FUNCTION_BLOCK TransferUnit (* Composite Function Block Type *)
  (* Standard: 61499-2 *)
  (* Version 0.0, 7/14/2016, Andrei, nxtControl GmbH, template *)
  PACKAGE Main;
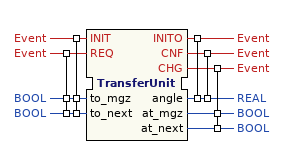
  EVENT_INPUT
    INIT WITH to_mgz, to_next; (* Initialization Request *)
    REQ WITH to_mgz, to_next; (* Normal Execution Request *)
  END_EVENT
  EVENT_OUTPUT
    INITO WITH angle; (* Initialization Confirm *)
    CNF WITH angle; (* Execution Confirmation *)
    CHG WITH at_mgz, at_next;
  END_EVENT
  VAR_INPUT
    to_mgz : BOOL; (* Input event qualifier *)
    to_next : BOOL;
  END_VAR
  VAR_OUTPUT
    angle : REAL; (* Output event qualifier *)
    at_mgz : BOOL;
    at_next : BOOL;
  END_VAR
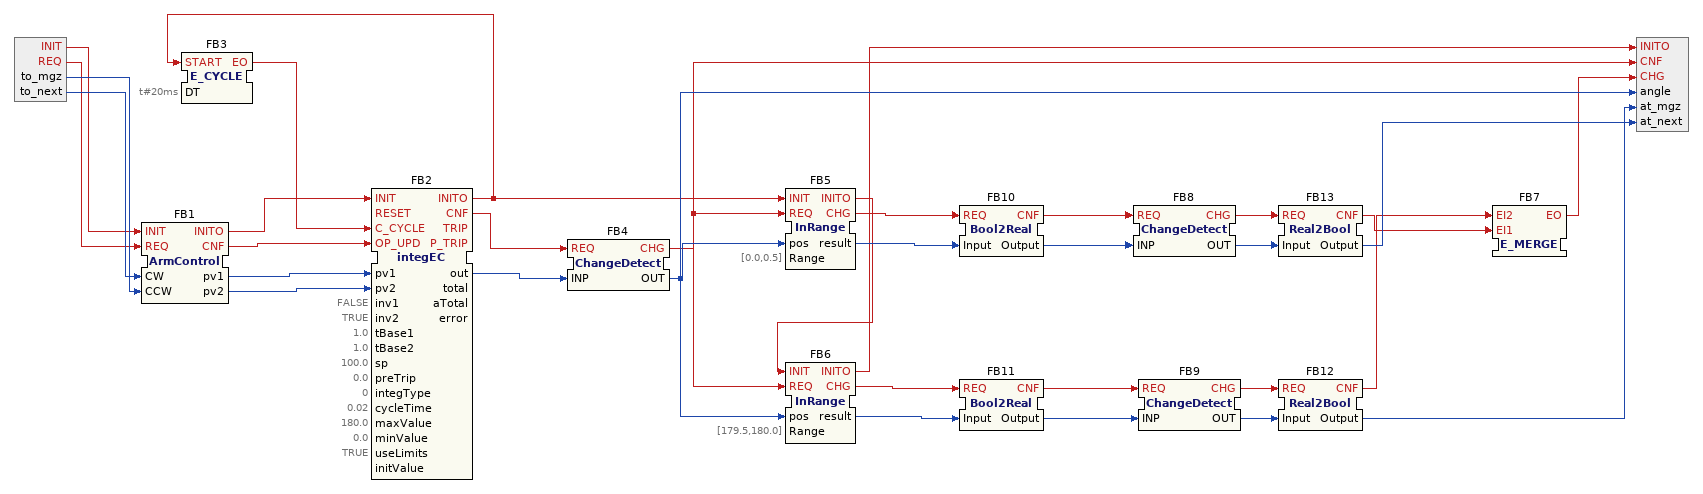
  FBS
    FB2 : integEC(inv1 := FALSE, inv2 := TRUE, tBase1 := 1.0, tBase2 := 1.0, sp := 100.0, preTrip := 0.0, integType := 0, cycleTime := 0.02, maxValue := 180.0, minValue := 0.0, useLimits := TRUE);
    FB3 : E_CYCLE(DT := t#20ms);
    FB4 : ChangeDetect;
    FB5 : InRange(Range := [0.0,0.5]);
    FB6 : InRange(Range := [179.5,180.0]);
    FB7 : E_MERGE;
    FB1 : ArmControl;
    FB8 : ChangeDetect;
    FB9 : ChangeDetect;
    FB10 : Bool2Real;
    FB11 : Bool2Real;
    FB12 : Real2Bool;
    FB13 : Real2Bool;
  END_FBS
  EVENT_CONNECTIONS
    REQ TO FB1.REQ;
    INIT TO FB1.INIT;
    FB1.CNF TO FB2.OP_UPD;
    FB1.INITO TO FB2.INIT;
    FB3.EO TO FB2.C_CYCLE;
    FB2.CNF TO FB4.REQ;
    FB2.INITO TO FB5.INIT;
    FB4.CHG TO FB5.REQ;
    FB5.INITO TO FB6.INIT;
    FB6.INITO TO INITO;
    FB7.EO TO CHG;
    FB4.CHG TO FB6.REQ;
    FB4.CHG TO CNF;
    FB2.INITO TO FB3.START;
    FB5.CHG TO FB10.REQ;
    FB6.CHG TO FB11.REQ;
    FB8.CHG TO FB13.REQ;
    FB12.CNF TO FB7.EI2;
    FB10.CNF TO FB8.REQ;
    FB11.CNF TO FB9.REQ;
    FB9.CHG TO FB12.REQ;
    FB13.CNF TO FB7.EI1;
  END_CONNECTIONS
  DATA_CONNECTIONS
    to_next TO FB1.CW;
    to_mgz TO FB1.CCW;
    FB1.pv1 TO FB2.pv1;
    FB1.pv2 TO FB2.pv2;
    FB2.out TO FB4.INP;
    FB4.OUT TO FB5.pos;
    FB4.OUT TO FB6.pos;
    FB4.OUT TO angle;
    FB5.result TO FB10.Input;
    FB6.result TO FB11.Input;
    FB9.OUT TO FB12.Input;
    FB8.OUT TO FB13.Input;
    FB10.Output TO FB8.INP;
    FB11.Output TO FB9.INP;
    FB12.Output TO at_mgz;
    FB13.Output TO at_next;
  END_CONNECTIONS
END_FUNCTION_BLOCK
